Fanuc KAREL source: compact_preamble.KL

PROGRAM KB00080
%NOLOCKGROUP
%ENVIRONMENT IOSETUP
VAR
P1:INTEGER;P2:INTEGER;P3:INTEGER;P4:INTEGER;P5:INTEGER;P6:INTEGER;P7:INTEGER;P8:INTEGER
BEGIN
P1=1
P2=1
P3=1
P4=1
P5=1
P6=1
P7=1
P8=1
GET_PORT_ASG(P1,P2,P3,P4,P5,P6,P7,P8)
END KB00080
